Staubli VAL3: commandExecute.pgx

program commandExecute(num& nArgs[] (dimensions=1), num nNbArgs (dimensions=1), string& sBuffer (dimensions=1), string sCommand (dimensions=1))
  local num nGetArg1
  local num nGetArg2
begin
  //execute command stored in global variables
  //bFlag check must be done previously in start()
  //popUpMsg(sCommand)
  switch sCommand
    case "gripper"
      call MX1_COMMANDS:gripper(nArgs[0])
      sBuffer="ACK: "+sCommand+" "+toString("",nArgs[0])
    break
    case "pickTool"
      call MX1_COMMANDS:changeToolMove(nArgs[0])
      sBuffer="ACK: "+sCommand+" "+toString("",nArgs[0])
    break
    case "power"
      call MX1_COMMANDS:power(nArgs[0])
      sBuffer="ACK: "+sCommand+" "+toString("",nArgs[0])
    break
    case "stopMove"
      call MX1_COMMANDS:stopMove()
      //stopMove()
      sBuffer="ACK: "+sCommand
    break
    case "restartMove"
      call MX1_COMMANDS:restartMove()
      //restartMove()
      sBuffer="ACK: "+sCommand
    break
    case "deleteMove"
      call MX1_COMMANDS:deleteMove()
      sBuffer="ACK: "+sCommand
    break
    case "isSettled"
      call MX1_COMMANDS:isSettled(nGetArg1)
      //bGetArg1 = isSettled()
      sBuffer="ACK: "+sCommand+" "+toString("",nGetArg1)
    break
    case "setFrame"
      call MX1_COMMANDS:setFrame(nArgs[0])
      sBuffer="ACK: "+sCommand+" "+toString("",nArgs[0])
    break
    case "setTool"
      call MX1_COMMANDS:setTool(nArgs[0])
      sBuffer="ACK: "+sCommand+" "+toString("",nArgs[0])
    break
    case "moveX"
      call MX1_COMMANDS:moveX(nArgs[0])
      sBuffer="ACK: "+sCommand+" "+toString(".3",nArgs[0])
    break
    case "moveY"
      call MX1_COMMANDS:moveY(nArgs[0])
      sBuffer="ACK: "+sCommand+" "+toString(".3",nArgs[0])
    break
    case "moveZ"
      call MX1_COMMANDS:moveZ(nArgs[0])
      sBuffer="ACK: "+sCommand+" "+toString(".3",nArgs[0])
    break
    case "getX"
      call MX1_COMMANDS:getX(nGetArg1)
      sBuffer="ACK: "+sCommand+" "+toString(".3",nGetArg1)
    break
    case "getY"
      call MX1_COMMANDS:getY(nGetArg1)
      sBuffer="ACK: "+sCommand+" "+toString(".3",nGetArg1)
    break
    case "getZ"
      call MX1_COMMANDS:getZ(nGetArg1)
      sBuffer="ACK: "+sCommand+" "+toString(".3",nGetArg1)
    break
    default
      logMsg("commandExecute fail: "+sCommand)
    break
  endSwitch
end
